(* IEC 61131-3 sources: AXOpen/src/inspectors/ctrl/src/AxoAnalogueInspector, 3 files *)

(* ---- IAxoAnalogueInspector.st ---- *)
USING AXOpen.Core;
NAMESPACE AXOpen.Inspectors
    INTERFACE IAxoAnalogueInspector

        METHOD Inspect : IInspector
            VAR_INPUT
                _parent : AXOpen.Core.IAxoObject;
                inData : REF_TO AxoAnalogueInspectorData;
                Status : LREAL;
            END_VAR
        END_METHOD

    END_INTERFACE
END_NAMESPACE

(* ---- AxoAnalogueInspector.st ---- *)
NAMESPACE AXOpen.Inspectors

    /// <summary>
    /// Class representing inspection of value within an interval.
    /// </summary>
    {S7.extern=ReadWrite}
    CLASS AxoAnalogueInspector EXTENDS AxoInspector IMPLEMENTS IAxoAnalogueInspector

        VAR PUBLIC
            // result data of inspection
            {#ix-attr:[RenderIgnore()]}
            _lastOutValue : LREAL;
        END_VAR

        VAR PRIVATE
            _data : REF_TO AxoAnalogueInspectorData;
        END_VAR

        /// <summary>
        /// Inspection method, which contains main logic of inspection.
        /// </summary>
        METHOD PUBLIC Inspect : IInspector
            VAR_INPUT
                _parent : AXOpen.Core.IAxoObject;
                inData : REF_TO AxoAnalogueInspectorData;
                Status : LREAL;
            END_VAR

            VAR
                tmpResult : BOOL;
                _minimum : LREAL;
                _value : LREAL;
                _maximum : LREAL;
            END_VAR

            VAR CONSTANT
                epsilon : REAL := 10000;
            END_VAR

            _data := inData;

            THIS.Initialize(_parent);
            _inspectorTask.Initialize(_parent);

            //return this instance
            Inspect := THIS;

            // pass address of data to set an inspection data
            _inspectorTask.SetInspectionData(_data);

            //check for overinspection
            IF(THIS.IsOverInspected())THEN
                RETURN;
            END_IF;

            //initialize and invoke inspector task
            _inspectorTask.Invoke();

            //do inspection
            IF (_inspectorTask.Execute()) THEN
                IF (_data^.IsByPassed) THEN
                    _data^.Result    := eInspectorResult#Bypassed;
                    _data^.TimeStamp := THIS.GetContext().GetRtc().NowUTC();
                    _inspectorTask.DoneWhen(TRUE);
                    RETURN;
                END_IF;

                _data^.Result := eInspectorResult#Running;

                _minimum := (_data^.RequiredMin * epsilon);
                _value := (Status * epsilon);
                _maximum := (_data^.RequiredMax * epsilon);

                _data^.DetectedStatus := Status;

                tmpResult := (_minimum <= _value) AND (_maximum >= _value);

                IF(NOT tmpResult) THEN
                    _lastOutValue := Status;
                END_IF;

                _inspectorTask._failTimer.OnDelay(THIS.GetContext(), TRUE, _data^.FailTime);
                _inspectorTask._passTimer.OnDelay(THIS.GetContext(), tmpResult, _data^.PassTime);

                IF(_inspectorTask._passTimer.output OR _inspectorTask._failTimer.output) THEN
                    _inspectorTask.DoneWhen(TRUE);
                    IF (_data^.Result = eInspectorResult#Failed) THEN
                        _data^.DetectedStatus := _lastOutValue;
                    END_IF;
                    THIS.OnDone();
                END_IF;
            END_IF;
        END_METHOD

        ///<summary>
        /// Set coordinator to this instance
        ///</summary>
        METHOD PUBLIC WithCoordinator : IAxoAnalogueInspector
            VAR_INPUT
                inCoordinator : AXOpen.Core.IAxoCoordinator;
            END_VAR

            _coordinator := inCoordinator;
            THIS._WithCoordinator(inCoordinator);

            WithCoordinator := THIS;
        END_METHOD

        ///<summary>
        /// If inspection fails, set result to data
        ///</summary>
        METHOD OnDone
        ;
        END_METHOD

        ///<summary>
        /// Set coordinator to this instance
        ///</summary>
        METHOD PUBLIC Data : REF_TO AxoAnalogueInspectorData

            Data := _data;
        END_METHOD
    END_CLASS
END_NAMESPACE

(* ---- AxoAnalogueInspectorData.st ---- *)
NAMESPACE AXOpen.Inspectors

    ///<summary>
    /// Data subjected to each analogue inspector instance.
    ///</summary>
    {S7.extern=ReadWrite}
    CLASS AxoAnalogueInspectorData EXTENDS AxoInspectorData
        VAR PUBLIC
            // <AxoAnalogueInspectorDataDeclaration>
            {#ix-set:AttributeName = "<#Min#>"}
            RequiredMin : LREAL;

            {#ix-attr:[ReadOnly()]}
            {#ix-set:AttributeName = "<#Detected#>"}
            DetectedStatus : LREAL;

            {#ix-set:AttributeName = "<#Max#>"}
            RequiredMax: LREAL;
            // </AxoAnalogueInspectorDataDeclaration>
        END_VAR
    END_CLASS
END_NAMESPACE
